PROGRAM pouStation1
VAR
END_VAR

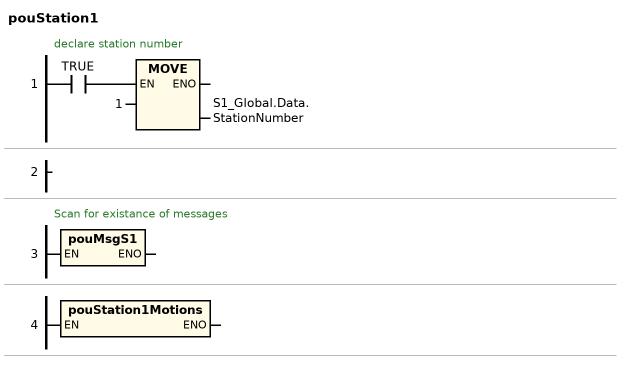
// NETWORK 1
// declare station number
S1_Global.Data.StationNumber := 1;

// NETWORK 2

// NETWORK 3
// Scan for existance of messages
pouMsgS1();

// NETWORK 4
pouStation1Motions();

END_PROGRAM

(* stored: Version 1.1.0.1, ProductVersion 3.1.4024.12
   POU pouStation1: Id {cbb126a5-ed47-44bc-850e-38b5e1137b4b}, SpecialFunc None *)
